Universal Robots PolyScope program: From_kettle_to_home.urp

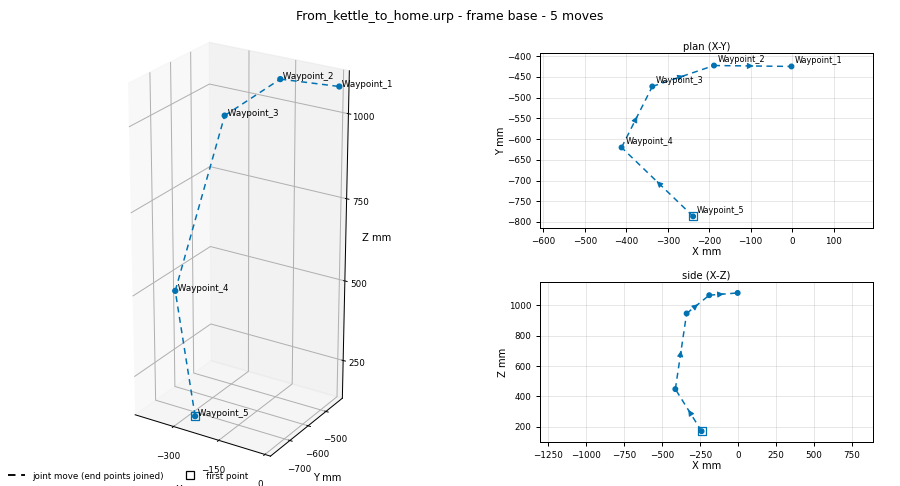
[picture p0: tool path of From_kettle_to_home.urp in frame base, 5 of 5 moves have a stored position in this frame; points joined in program order, loops and branches not executed]
Program From_kettle_to_home (installation=default directory=/programs/Matcha createdIn=5.12.6.1102099 lastSavedIn=5.12.6.1102099 robotSerialNumber=20215500597)
Calibrated DH parameters: a=[0.000193, -0.066673, -0.391568, -0.000012, 0.00005, 0]; d=[0.162643, -472.05677, 465.132521, 7.058239, 0.099746, 0.099582]; alpha=[1.571116, 0.00089, 0.003862, 1.569269, -1.569248, 0]; deltaTheta=[0, -1.413394, 7.628392, 0.068187, 0, -0.000001]
Robot Program (runOnlyOnce=true)
  MoveJ speed 60 deg/s, acceleration 80 deg/s^2 (useActiveTCP=true) feature=Base
    Waypoint Waypoint_5: TCP in base x=-238.817 y=-786.483 z=171.154 mm, rx=0.0286 ry=-2.2144 rz=2.2271 rad; joints [49.901, -56.995, 96.504, -40.113, 49.291, 179.676] deg; TCP offset x=0 y=0 z=191.5 mm, rx=0 ry=0 rz=0 rad
    Waypoint Waypoint_4: TCP in base x=-411.417 y=-620.304 z=448.013 mm, rx=0.5178 ry=-2.1305 rz=2.1802 rad; joints [22.119, -66.389, 66.781, 0.117, 10.43, 163.845] deg
    Waypoint Waypoint_3: TCP in base x=-337.24 y=-473.129 z=945.528 mm, rx=1.5856 ry=0.1092 rz=0.0753 rad; joints [7.565, -80.223, 27.532, -72.21, -1.151, 123.731] deg
    Waypoint Waypoint_2: TCP in base x=-188.417 y=-422.615 z=1065.641 mm, rx=1.0298 ry=1.2726 rz=-1.2396 rad; joints [0.065, -82.209, 8.1, -73.224, 7.414, 51.58] deg
    Waypoint Waypoint_1: TCP in base x=-1.55 y=-424.818 z=1080.554 mm, rx=-0.0044 ry=-2.2186 rz=2.2204 rad; joints [0.002, -89.997, -0.002, -89.999, 0, 0.001] deg
